Staubli VAL3: clkCleanupChuck1.pgx

program clkCleanupChuck1()
  local num nAirexIdx
begin
  switchMagnet=false
  statusCleanupChuck1 = colorRunning

  call selectedCheck()
  call print("cleanup (airex) start")

  // -- pick vacuum chuck1's and put them back to their original place
  for nAirexIdx=0 to 5
    if !bSelectItem or (bSelectedItems[nAirexIdx]==true)
      call print("put away chuck " + toString("1.0", nAirexIdx))
      // -- move over final airex position (where the chuck is from gluing) and down
      // -- for edge positions make a curve to avoid hitting side bar
      if nAirexIdx == 0 or nAirexIdx == 3
        movej(appro(airexInitial[1], trZsafe), tTool, mFast)
      endIf

      call moveDown(airexFinal[nAirexIdx], mSlow, trZero, false)

      // -- lift chuck1
      switchMagnet=true
      delay(waitShort)
      movel(appro(airexFinal[nAirexIdx], trZsafe), tTool, mSlow)
      //waitEndMove()

      // -- move over/to initial chuck position
      // -- for edge positions make a curve to avoid hitting side bar
      if nAirexIdx == 0 or nAirexIdx == 3
        movej(appro(airexInitial[1], trZsafe), tTool, mFast)
      endIf
      call moveDown(chuck1[nAirexIdx], mSlow, trZero, false)

      // -- release it
      switchMagnet=false

      // -- move up
      movel(appro(chuck1[nAirexIdx], trZsafe), tTool, mSlow)
    endIf
  endFor

  // -- move back somewhere
  call print("parking robot")
  waitEndMove()
  movej(jInitialPosition, tTool, mFast)
  waitEndMove()
  statusCleanupChuck1 = colorOn
  statusDoAirex = colorGray
  call print("cleanup (airex) done")
  //call selectedClear()

end
